(* IEC 61131-3 sources: generating_plc_code_with_llms/Code#2/Platypus2/first run, 21 files *)

(* ---- 12.st ---- *)
// 64.78193426132202s
// 2
FUNCTION sinehyp(X)
    IF (X < 0.0) THEN
        RETURN -sinehyp(-X);
    END_IF
    IF (X > 1.0) THEN
        RETURN 1.0;
    END_IF
    IF (X == 0.0) THEN
        RETURN 0.0;
    END_IF
    IF (X < 1.0) THEN
        RETURN SQRT(2.0)*EXP(-X*X);
    ELSE
        RETURN EXP(X)-EXP(-X);
    END_IF
END_FUNCTION

(* ---- 15.st ---- *)
// 102.83285927772522s
// 2
FUNCTION FC1002 :BOOL
VAR_INPUT
	E_A, SENSOR: BOOL;
	ZEITW: TIME;
END_VAR
VAR_IN_OUT
	ZEIT:TON;
	P_HU, P_AL: BOOL;
END_VAR
IF E_A THEN
	P_HU := FALSE;
	P_AL := FALSE;
	SENSOR := TRUE;
	WHILE SENSOR DO
		ZEITW := ZEIT + 3.0;
		IF ZEITW > TIME(1) THEN
			P_HU := TRUE;
		END_IF;
	END_WHILE;
	IF P_HU THEN
		P_AL := FALSE;
	ELSE
		P_AL := TRUE;
	END_IF;
ENDIF;
RETURN(P_HU);

(* ---- 18.st ---- *)
// 127.77234196662903s
// 2
FUNCTION FC1003 : VOID
VAR_INPUT
    IN_R:REAL;
    IN_MAX, IN_MIN:REAL;
    OUT_MAX, OUT_MIN:REAL;
END_VAR
VAR_OUTPUT
    OUT_R:REAL;
    FEH:BOOL;
END_VAR
VAR_TEMP
    DIFF1, DIFF2:REAL;
END_VAR

IF IN_R > IN_MAX THEN
    OUT_R := -999.0;
    FEH := TRUE;
ELSE IF IN_R < IN_MIN THEN
    OUT_R := -999.0;
    FEH := TRUE;
ELSE
    DIFF1 := (OUT_MAX - OUT_MIN) / (IN_MAX - IN_MIN);
    DIFF2 := (OUT_R - OUT_MIN) * DIFF1 + OUT_MIN;
    IF DIFF2 > OUT_MAX THEN
        OUT_R := -999.0;
        FEH := TRUE;
    ELSE
        OUT_R := DIFF2;
    END_IF
ENDIF

(* ---- 21.st ---- *)
// 862.7894697189331s
// 2
FUNCTION BURNER(IN, STAGE2, OVER_TEMP, OIL_TEMP, FLAME, RST, RST_TIMER, PRE_HEAT_TIME, PRE_VENT_TIME, PRE_IGNITE_TIME, POST_IGNITE_TIME, STAGE2_DELAY, SAFETY_TIME, LOCKOUT_TIME, MULTIPLE_IGNITION, KW1, KW2)
    IF IN THEN
        STATUS := 110;
        PRE_HEAT := TRUE;
        RST_TIMER := FALSE;
        OIL_TEMP := FALSE;
        FLAME := FALSE;
        CYCLES := 0;
    END_IF
    IF (PRE_HEAT) THEN
        STATUS := 111;
        PRE_HEAT := FALSE;
        RST_TIMER := TRUE;
        OIL_TEMP := FALSE;
        FLAME := FALSE;
        CYCLES := 0;
    END_IF
    IF (OIL_TEMP) THEN
        STATUS := 112;
        PRE_HEAT := FALSE;
        RST_TIMER := TRUE;
        OIL_TEMP := FALSE;
        FLAME := FALSE;
        CYCLES := 0;
    END_IF
    IF (FLAME) THEN
        STATUS := 113;
        PRE_HEAT := FALSE;
        RST_TIMER := TRUE;
        OIL_TEMP := FALSE;
        FLAME := FALSE;
        CYCLES := 0;
    END_IF
    IF (RST) THEN
        STATUS := 110;
        PRE_HEAT := FALSE;
        RST_TIMER := TRUE;
        OIL_TEMP := FALSE;
        FLAME := FALSE;
        CYCLES := 0;
    END_IF
    IF (RST_TIMER) THEN
        STATUS := 110;
        PRE_HEAT := TRUE;
        RST_TIMER := FALSE;
        OIL_TEMP := FALSE;
        FLAME := FALSE;
        CYCLES := 0;
    END_IF
    IF (PRE_HEAT) THEN
        STATUS := 111;
        PRE_HEAT := FALSE;
        RST_TIMER := TRUE;
        OIL_TEMP := FALSE;
        FLAME := FALSE;
        CYCLES := 0;
    END_IF
    IF (OIL_TEMP) THEN
        STAT TIME :=  STAT t1111111111111111111111111111111111110;
        STAT OIL_IF (OIL_IF (STATUS :=  IF (PRE_IF (RUNTIL_IF (IF (OIL_IF (OIL_IF (OIL_IF (IF (OIL_IF (OIL_IF (OIL_IF (OIL_IF (OIL_IF (OIL_IF (
        STAT TIME :=  IF (PRE_IF (STATUS :=  IF (RUNTIL_IF (OIL_IF (OIL_IF (OIL_IF (OIL_IF (OIL_IF (OIL_IF (IF (OIL_IF (OIL_IF (
        STAT TIME :=  IF (PRE_IF (STATUS :=  STAT t10.
        STAT TX :=  IF (RUNTIL_IF (OIL_IF (OIL_IF (OIL_IF (OIL_IF (OIL_IF (OIL_IF (OIL_IF (OIL_IF (PRE_IF (STATUS :=  IF (OIL_IF (
        STAT TIME :=  IF (RUNTIL_IF (STATE :=  STAT TX :=  IF (OIL_IF (OIL_IF (IF (PRE_IF (OIL_IF (OIL_IF (OIL_IF (STATUS :=  IF (OIL_IF (
        STAT t10.
        STAT TIME :=  STAT TX :=  IF (RUNTIL_IF (OIL_IF (OIL_IF (PRE_IF (OIL_IF (OIL_IF (OIL_IF (STATUS :=  IF (OIL_IF (OIL_IF (
        STAT t10.
        STAT TIME :=  IF (RUNTIL_IF (OIL_IF (OIL_IF (PRE_IF (IF (IF (IF (OIL_IF (STATUS :=  IF (OIL_IF (OIL_IF (OIL_IF (OIL_IF (
        STAT TIME :=  IF (RUNTIL_IF (IF (IF (OIL_IF (PRE_IF (OIL_IF (OIL_IF (OIL_IF (STATUS :=  IF (OIL_IF (OIL_IF (OIL_IF (OIL_IF (
        STAT TIME :=  IF (RUNTIL_IF (OIL_IF (PRE_IF (OIL_IF (OIL_IF (OIL_IF (STATUS :=  STAT t10.
        STATOMITERLATE_IF (OIL_IF (OIL_IF (OIL_IF (RUNTIL_IF (OIL_IF (PRE_IF (OIL_IF (OIL_IF (OIL_IF (STATUS :=  IF (OIL_IF (OIL_IF (
        STAT TIME :=  IF (OIL_IF (OIL_IF (RUNTIL_IF (OIL_IF (PRE_IF (STARET10.
        STAT t11111111111111111111111111111111111111111111111111111111110.
        STAT TIME :=  IF (IF (OIL_IF (PRE_IF (STATUS :=  IF (RUNTIL_IF (OIL_IF (OIL_IF (OIL_IF (OIL_IF (OIL_IF (IF (IF (OIL_IF (OIL_IF (OIL_IF (OIL_IF (OIL_IF (STATUS :=  IF (PRE_IF (RUNTIL_IF (
        STAT TIME :=  IF (OIL_IF (OIL_IF (OIL_IF (OIL_IF (OIL_IF (OIL_IF (OIL_IF (OIL_IF (STATUS :=  IF (PRE_IF (RUNTIL_IF (
        STAT TIME :=  IF (OIL_IF (OIL_IF (OIL_IF (OIL_IF (OIL_IF (OIL_IF (OIL_IF (OIL_IF (STATUS :=  STAT t10.
        STAT TX :=  IF (PRE_IF (RUNTIL_IF (IF (OIL_IF (OIL_IF (OIL_IF (OIL_IF (OIL_IF (OIL_IF (OIL_IF (STATUS :=  IF (OIL_IF (IF (IF (
        STAT TIME :=  IF (PRE_IF (RUNTIL_IF (OIL_IF (PRE_IF (OIL_IF (OIL_IF (OIL_IF (OIL_IF (OIL_IF (STATUS :=  STAT t10.
        STAT TX :=  IF (OIL_IF (OIL_IF (RUNTIL_IF (OIL_IF (PRE_IF (OIL_IF (OIL_IF (OIL_IF (OIL_IF (OIL_IF (STATUS :=  IF (OIL_IF (IF (OIL_IF (OIL_IF (OIL_IF (RUNTIL_IF (OIL_IF (PRE_IF (
        STAT TIME :=  IF (OIL_IF (OIL_IF (OIL_IF (STATUS :=  STAT TX :=  IF (OIL_IF (IF (OIL_IF (OIL_IF (RUNTIL_IF (OIL_IF (PRE_IF (OIL_IF (OIL_IF (
        STAT t10.
        STAT TIME :=  STAT TX :=  IF (STATUS :=  IF (IF (OIL_IF (OIL_IF (RUNTIL_IF (OIL_IF (PRE_IF (OIL_IF (OIL_IF (OIL_IF (O

(* ---- 19.st ---- *)
// 154.3342866897583s
// 2
FUNCTION_BLOCK FB1005
VAR_INPUT
    START:BOOL;
    DICKE, V_MAX, V_MIN:REAL;
END_VAR
VAR_OUTPUT
    D_MAX, D_MIN:REAL;
    P1:BOOL;
END_VAR
VAR
    FO:BOOL;
END_VAR
IF START THEN
    DICKE := 0.0;
    V_MAX := 0.0;
    V_MIN := 0.0;
    D_MAX := 0.0;
    D_MIN := 0.0;
    P1 := FALSE;
ELSE
    DICKE := 0.0;
    V_MAX := 0.0;
    V_MIN := 0.0;
    D_MAX := 0.0;
    D_MIN := 0.0;
    P1 := FALSE;
ENDIF
IF START THEN
    IF (DICKE > V_MAX) OR (DICKE < V_MIN) THEN
        P1 := TRUE;
    END_IF
ELSE
    IF (DICKE > V_MAX) OR (DICKE < V_MIN) THEN
        P1 := TRUE;
    END_IF
ENDIF
END_FUNCTION_BLOCK

(* ---- 1.st ---- *)
// 77.3076605796814s
// 2
PROGRAM main

VAR
	xAllOn : BOOL;
	xAllOff : BOOL;

	xAlarm1 : BOOL;
    xAlarm2 : BOOL;
END_VAR

BEGIN
	xAllOn := TRUE;
	xAllOff := FALSE;

	xAlarm1 := TRUE;
    xAlarm2 := FALSE;

	IF xAllOn THEN
		xAllOff := FALSE;
	ELSE
		xAllOff := TRUE;

	IF xAllOff THEN
		xAllOn := FALSE;
	ELSE
		xAllOn := TRUE;
END_PROGRAM

(* ---- 10.st ---- *)
// 69.50946974754333s
// 2
PROGRAM sigmoid;

VAR_OUTPUT
    Y : REAL;
END_VAR

VAR
    A : REAL := 1.0;
    B : REAL := 1.0;
    C : REAL := 1.0;
    D : REAL := 1.0;
    E : REAL := 1.0;
END_VAR

PROCEDURE sigmoid(X: REAL);
BEGIN
    Y := A * (1.0 / (1.0 + EXP(-B * X)));
END_PROCEDURE

VAR_INPUT
    X : REAL;
END_VAR

VAR
    Y : REAL;
END_VAR

Y := sigmoid(X);

(* ---- 11.st ---- *)
// 35.603342056274414s
// 2
PROGRAM sign;
VAR_INPUT
    x : REAL;
END_VAR
IF x > 0 THEN
    RETURN(1);
ELSE IF x < 0 THEN
    RETURN(-1);
ELSE
    RETURN(0);
ENDIF;

(* ---- 13.st ---- *)
// 116.2343533039093s
// 2
PROGRAM main;

VAR
    aNumbers : ARRAY[0..MAXNUMBERS] OF INT;
    nCnt : INT;
    i : INT;
    s : STRING(10);
END_VAR

BEGIN
    CLEAR_SCREEN;
    PRINT('Enter the number of random numbers:');
    READLN(nCnt);
    FOR i := 0 TO nCnt - 1 DO
        aNumbers[i] := RANDOM(0, 99);
    END_FOR;
    PRINT('The list contains the following numbers:');
    FOR i := 0 TO nCnt - 1 DO
        PRINT(aNumbers[i], ' ');
    END_FOR;
    REPEAT
        PRINT('Enter a number to search for:');
        READLN(s);
        IF s = '10' THEN
            EXIT;
        END_IF;
        FOR i := 0 TO nCnt - 1 DO
            IF aNumbers[i] = INT(s) THEN
                EXIT;
            END_IF;
        END_FOR;
    UNTIL FALSE;
    PRINT('The number was not found.');
END main.

(* ---- 14.st ---- *)
// 42.977917194366455s
// 2
IF MEW > SP THEN
	OUT := TRUE;
ELSE IF MEW < SP - HYS * SP THEN
	OUT := FALSE;
END_IF;

(* ---- 16.st ---- *)
// 162.15188837051392s
// 2
PROGRAM main
    VAR
        North_green : BOOL;
        North_yellow : BOOL;
        North_red : BOOL;
        East_green : BOOL;
        East_yellow : BOOL;
        East_red : BOOL;
        T1 : TON;
    END_VAR

    NORTH_GREEN := TRUE;
    EAST_RED := FALSE;

    T1.INITIALIZE(10000);
    T1.START();

    WHILE (T1.RUNNING) DO
        IF (T1.ELAPSED() < 5000) THEN
            NORTH_GREEN := TRUE;
            EAST_RED := FALSE;
        ELSEIF (T1.ELAPSED() >= 5000 AND T1.ELAPSED() <= 9500) THEN
            NORTH_YELLOW := TRUE;
            EAST_GREEN := TRUE;
        ELSEIF (T1.ELAPSED() > 9500 AND T1.ELAPSED() < 10000) THEN
            NORTH_RED := TRUE;
            EAST_YELLOW := TRUE;
        END_IF;
    END_WHILE;
END_PROGRAM main

(* ---- 17.st ---- *)
// 70.54809927940369s
// 2
IF (aiOutside < 18) THEN
    sShowText := "Cold";
ELSIF (aiOutside >= 18 AND aiOutside <= 25) THEN
    IF (aiHumidity BETWEEN 40 AND 75) THEN
        sShowText := "Opt";
    ELSE
        sShowText := "Temp. OK";
ELSE
    sShowText := "Hot";
END_IF;

(* ---- 2.st ---- *)
// 86.31310868263245s
// 2
PROGRAM binomial_coefficient;

VAR_INPUT
    N : INT;
    K : INT;
    i : INT;
END_VAR

BEGIN
    WRITE(N, 'Enter the number of elements in the set:');
    READLN(N);
    WRITE(K, 'Enter the number of elements to choose from the set:');
    READLN(K);

    i := 1;
    WHILE (i <= K) DO
        IF (i MOD 2 = 0) THEN
            WRITE(' ', N - i + 1, '!', '/', i, '=', i * (N - i));
        ELSE
            WRITE(' ', N - i + 1, '!', '/', i, '=', (i - 1) * (N - i));
        END_IF;
        INC(i);
    END_WHILE;
END_PROGRAM.

(* ---- 20.st ---- *)
// 51.82499980926514s
// 2
IF I1 THEN
    IF I2 THEN
        WAIT TL
    ELSE
        Q1 := TRUE
    END_IF
ELSE
    IF NOT I2 THEN
        WAIT TL
    ELSE
        Q2 := TRUE
    END_IF
END_IF

(* ---- 3.st ---- *)
// 66.81055355072021s
// 2
PROGRAM fibunacci
VAR_INPUT
    X : INT;
END_VAR
VAR
    t1 : DINT;
    t2 : DINT;
    x_tmp : INT;
END_VAR
IF X = 0 THEN
    RETURN(0);
ELSE IF X = 1 THEN
    RETURN(1);
ELSE
    t1 := 0;
    t2 := 1;
    WHILE t1 < X DO
        x_tmp := t1 + t2;
        t1 := t2;
        t2 := x_tmp;
    END_WHILE;
    RETURN(t2);
ENDIF;

(* ---- 4.st ---- *)
// 54.82225155830383s
// 2
IF (aiLevel < 1) THEN
    DO_ALARM := TRUE;
ELSEIF (aiLevel > 99) THEN
    DO_HIGH := TRUE;
ELSEIF (aiLevel > 50) THEN
    DO_OK := TRUE;
ELSEIF (aiLevel < 10) THEN
    DO_LOW := TRUE;
END_CASE;

(* ---- 5.st ---- *)
// 151.2458050251007s
// 2
PROGRAM GateController;

VAR
    Start_Loop : BOOL := FALSE;
    one_hour : TIME := T#1h;
    One_Hour_Timer : TON;
    Gate_Open : BOOL := FALSE;
    Close_Gate_Inst : BOOL := FALSE;
    Sensed_Car : BOOL := FALSE;
    Sensed_Car_Inst : BOOL := FALSE;
    Sensed_App : BOOL := FALSE;
    Mobile_Inst : BOOL := FALSE;
    Auth : STRING := 'abcd';
    my_defined_str : STRING := 'abcd';
END_VAR

BEGIN
    IF Start_Loop THEN
        WHILE TRUE DO
            IF Gate_Open THEN
                CLOSE_GATE;
                Close_Gate_Inst := TRUE;
            END_IF;
            IF Sensed_Car THEN
                OPEN_GATE;
                Sensed_Car_Inst := TRUE;
            END_IF;
            IF Sensed_App THEN
                OPEN_GATE;
                Sensed_App_Inst := TRUE;
            END_IF;
            IF Close_Gate_Inst OR Sensed_Car_Inst OR Sensed_App_Inst THEN
                CLOSE_GATE;
                Gate_Open := FALSE;
            END_IF;
            IF TIMER_EXPIRED(One_Hour_Timer) THEN
                CLOSE_GATE;
                Gate_Open := FALSE;
            END_IF;
        END_WHILE;
    END_IF;
END_PROGRAM.

(* ---- 6.st ---- *)
// 225.8638265132904s
// 2
PROGRAM crane_lift
    VAR
        WAIT : UINT := 0;
        TOP_POSITION : UINT := 1;
        BOTTOM_POSITION : UINT := 2;
        GETBOX : UINT := 3;
        UNLOAD_POSITION : UINT := 4;
        UNLOAD_BOX : UINT := 5;
    END_VAR

    VAR
        (*-- digital outputs*)
        doConvTop: BOOL;
        doConvBottom: BOOL;
        doConvLift: BOOL;
        doLiftTop: BOOL;
        doLiftBottom: BOOL;
        doLiftUnload: BOOL;
        (*-- digital inputs*)
        diConvTop: BOOL;
        diConvBottom: BOOL;
        diLiftTop: BOOL;
        diLiftBottom: BOOL;
        diLiftUnload: BOOL;
        diBoxLift: BOOL;
        (*-- status variables*)
        selectLift: UINT;
        ConvTopOn: BOOL;
        ConvBottomOn: BOOL;
    END_VAR

    (*-- digital outputs*)
    doConvTop := FALSE;
    doConvBottom := FALSE;
    doConvLift := FALSE;
    doLiftTop := FALSE;
    doLiftBottom := FALSE;
    doLiftUnload := FALSE;
    (*-- digital inputs*)
    diConvTop := FALSE;
    diConvBottom := FALSE;
    diLiftTop := FALSE;
    diLiftBottom := FALSE;
    diLiftUnload := FALSE;
    diBoxLift := FALSE;
    (*-- status variables*)
    selectLift := 0;
    ConvTopOn := FALSE;
    ConvBottomOn := FALSE;

    WHILE TRUE DO
        WAIT := WAIT + 1;
        IF (WAIT > 25) THEN
            (*-- digital outputs*)
            doConvTop := NOT doConvTop;
            doConvBottom := NOT doConvBottom;
            doL

(* ---- 7.st ---- *)
// 81.30413317680359s
// 2
PROGRAM Crane
    VAR
        CONSTANT
            MAX_INDEX : USINT := 4;
        aWeights : ARRAY[0..MAX_INDEX] OF INT;
        iCnt : USINT;
        sumWeight : DINT;
        avgWeight : INT;
    END_VAR
    PROCESS
        FOR iCnt := 0 TO MAX_INDEX - 1 DO
            aWeights[iCnt] := INPUT(0);
        END_FOR
        sumWeight := SUM(aWeights, MAX_INDEX);
        avgWeight := sumWeight / MAX_INDEX;
    END_PROCESS
END_PROGRAM

(* ---- 8.st ---- *)
// 102.14219069480896s
// 2
PROGRAM lambertw
VAR
    X : REAL;
    i : INT;
    we : REAL;
    w1e : REAL;
    ewx : REAL;
    last : DWORD;
END_VAR

IF (X > 0) THEN
    RETURN
ELSE
    X := -X;
ENDIF

FOR i := 1 TO 200 STEP 5 DO
    w := 0.0;
    we := 1.0 / X;
    ewx := EXP(we);
    FOR j := 1 TO 200 STEP 5 DO
        IF (j > i) THEN
            IF (ewx < 1.0) THEN
                w1e := we * ewx;
                IF (w1e >= 1.0) THEN
                    RETURN
                END_IF
                w := w + w1e / j;
            ELSE
                RETURN
            END_IF
        END_IF
    NEXT
ENDFOR
X := -X * LOG(w);
END_PROGRAM

(* ---- 9.st ---- *)
// 52.79196882247925s
// 2
IF (YEAR MOD 4 = 0) THEN
    IF (YEAR MOD 100 = 0) THEN
        IF (YEAR MOD 400 = 0) THEN
            PRINT "Year is a leap year"
        ELSE
            PRINT "Year is not a leap year"
        END_IF
    ELSE
        PRINT "Year is not a leap year"
    END_IF
ELSE
    PRINT "Year is not a leap year"
END_IF
